// TIA Portal V17 export
// export: Created 2021-12-03T08:13:15.0467151Z, ExportSetting WithDefaults, DisplayName Totally Integrated Automation Portal, DisplayVersion V17, DisplayName TIA Portal Openness, DisplayVersion V17, DisplayName TIA Portal Version Control Interface, DisplayVersion V17, DisplayName STEP 7 Professional, DisplayVersion V17, DisplayName STEP 7 Safety, DisplayVersion V17, DisplayName WinCC Advanced, DisplayVersion V17
DATA_BLOCK "FGDB_Inputs"   // DB50, F_DB
VERSION : 0.1
// stored: AutoNumber false
   VAR
      "I_/EmStpAccCon_Ch1" : Bool;   // Консоль ускорителя канал 1
      "I_/EmStpP1_Ch1" : Bool;   // Пульт Р1 канал 1
      "I_/EmStpP2_Ch1" : Bool;   // Пульт Р2 канал 1
      I_PrDoor1Cls_Ch1 : Bool;   // Замок блокирующий дверь 1 канал 1
      I_PrDoor2Cls_Ch1 : Bool;   // Замок блокирующий дверь 2 канал 1
      I_Spare40_5 : Bool;   // Spare
      "I_/EmStpDosimeter_Ch1" : Bool;   // Дозиметр канал 1
      I_PrDoor1Req : Bool;   // Запрос на открытие двери 1
      I_P3AckInSArea_Ch1 : Bool;   // Сброс внутри периметра безопасности
      I_FBPowerModulator : Bool;   // Обратная связь модулятора
      I_FBPowerConveyor : Bool;   // Обратная связь частотного преобразователя
      I_FBPowerXRayUnit : Bool;   // Обратная связь ускоритель
      "I_/EmStpAccCon_Ch2" : Bool;   // Консоль ускорителя канал 2
      "I_/EmStpP1_Ch2" : Bool;   // Пульт Р1 канал 2
      "I_/EmStpP2_Ch2" : Bool;   // Пульт Р2 канал 2
      I_PrDoor1Cls_Ch2 : Bool;   // Замок блокирующий дверь 1 канал 2
      I_PrDoor2Cls_Ch2 : Bool;   // Замок блокирующий дверь 2 канал 2
      I_Spare42_2 : Bool;   // Spare
      "I_/EmStpDosimeter_Ch2" : Bool;   // Дозиметр канал 2
      I_PrDoor2Req : Bool;   // Запрос на открытие двери 2
      I_P1AckEmStpOutSArea : Bool;   // Сброс снаружи периметра безопасности
      I_FBPowerChiller : Bool;   // Обратная связь чиллер
      I_FBPower_AccConsol : Bool;   // Обратная связь консоль ускорителя
      I_FBPowerModulator1P : Bool;   // Обратная связь модулятора 1 фаза
      "I_/EmStpP3_Ch1" : Bool;   // Пульт P3 канал 1
      I_P2AgreeBut_Ch1 : Bool;   // Кнопка разрешения канал 1
      I_Spare60_2 : Bool;   // Spare
      I_Spare60_3 : Bool;   // Spare
      I_Spare60_4 : Bool;   // Spare
      I_Spare60_5 : Bool;   // Spare
      I_Spare60_6 : Bool;   // Spare
      I_Spare60_7 : Bool;   // Spare
      I_P1KeyGenRel_Ch1 : Bool;   // Главный ключ разрешения канал 1
      I_P1KeyAccRel_Ch1 : Bool;   // Ключ разрешения включения ускорителя канал 1
      I_Spare61_2 : Bool;   // Spare
      I_Spare61_3 : Bool;   // Spare
      "I_/EmStpP3_Ch2" : Bool;   // Пульт P3 канал 2
      I_P2AgreeBut_Ch2 : Bool;   // Кнопка разрешения канал 2
      I_Spare61_6 : Bool;   // Spare
      I_Spare61_7 : Bool;   // Spare
      I_Spare62_0 : Bool;   // Spare
      I_Spare62_1 : Bool;   // Spare
      I_Spare62_2 : Bool;   // Spare
      I_Spare62_3 : Bool;   // Spare
      I_P1KeyGenRel_Ch2 : Bool;   // Главный ключ разрешения канал 2
      I_P1KeyAccRel_Ch2 : Bool;   // Ключ разрешения включения ускорителя канал 2
      I_Spare62_6 : Bool;   // Spare
      I_Spare62_7 : Bool;   // Spare
   END_VAR
BEGIN
END_DATA_BLOCK
